# EPICS substitutions: apps/plcApp/Db/torus_comm.substitutions
#
# torus_comm.substitutions
#
# Author: Wesley Moore (wmoore@jlab.org)
# Date:   June 2017
#

file "db/torus_bi_generic.db" { pattern
    { PLCID,     P,        R,    TAG,            ZNAM,  ONAM,       ZSV,        OSV,    DESC }
    { PLC_TORUS, B_TORUS:, MPS:, UPS_On_Battery, Ok,    Warning,    NO_ALARM,   MAJOR,  "PLC On UPS Battery" }
}
